FUNCTION F_Delete_ST_AnyType : HResult
VAR_INPUT
	name : STRING(80);
	varType : MPM_JsonParser.E_TypeClassEx;
END_VAR
VAR_IN_OUT
	stAnyType : MPM_JsonParser.ST_AnyType_User;
END_VAR
VAR
	pPointer_BYTE : POINTER TO BYTE;
	pPointer_BOOL : POINTER TO BOOL;
	pPointer_LREAL : POINTER TO LREAL;
	pPointer_DINT : POINTER TO DINT;
	pPointer_LINT : POINTER TO LINT;	
	pPointer_UDINT : POINTER TO UDINT;	
	pPointer_INT : POINTER TO INT;		
	pPointer_REAL : POINTER TO REAL;
	pPointer_WORD : POINTER TO WORD;		
END_VAR

stAnyType.name := name;
stAnyType.typeclass := varType;
IF stAnyType.pvalue > 0 THEN
	F_Delete_ST_AnyType := MPM_FBResult.E_Result.S_FAILED;
	RETURN;
END_IF
CASE varType OF
	MPM_JsonParser.E_TypeClassEx.TYPE_BOOL:
		pPointer_BYTE := stAnyType.pvalue;
		stAnyType.diSize := SIZEOF(BOOL);
		F_Delete_ST_AnyType := MPM_FBResult.E_Result.S_OK;
	MPM_JsonParser.E_TypeClassEx.TYPE_BYTE:
		stAnyType.pvalue := __NEW(BYTE);	
		stAnyType.diSize := SIZEOF(BYTE);	
		F_Delete_ST_AnyType := MPM_FBResult.E_Result.S_OK;
	MPM_JsonParser.E_TypeClassEx.TYPE_LREAL:
		stAnyType.pvalue := __NEW(LREAL);	
		stAnyType.diSize := SIZEOF(LREAL);	
		F_Delete_ST_AnyType := MPM_FBResult.E_Result.S_OK;		
	MPM_JsonParser.E_TypeClassEx.TYPE_DINT:
		stAnyType.pvalue := __NEW(DINT);	
		stAnyType.diSize := SIZEOF(DINT);	
		F_Delete_ST_AnyType := MPM_FBResult.E_Result.S_OK;
	MPM_JsonParser.E_TypeClassEx.TYPE_LINT:
		stAnyType.pvalue := __NEW(LINT);	
		stAnyType.diSize := SIZEOF(LINT);
		F_Delete_ST_AnyType := MPM_FBResult.E_Result.S_OK;	
	MPM_JsonParser.E_TypeClassEx.TYPE_UDINT:
		stAnyType.pvalue := __NEW(UDINT);	
		stAnyType.diSize := SIZEOF(UDINT);
		F_Delete_ST_AnyType := MPM_FBResult.E_Result.S_OK;	
	MPM_JsonParser.E_TypeClassEx.TYPE_INT:
		stAnyType.pvalue := __NEW(INT);	
		stAnyType.diSize := SIZEOF(INT);
		F_Delete_ST_AnyType := MPM_FBResult.E_Result.S_OK;		
	MPM_JsonParser.E_TypeClassEx.TYPE_REAL:
		stAnyType.pvalue := __NEW(REAL);	
		stAnyType.diSize := SIZEOF(REAL);	
		F_Delete_ST_AnyType := MPM_FBResult.E_Result.S_OK;		
	MPM_JsonParser.E_TypeClassEx.TYPE_WORD:
		stAnyType.pvalue := __NEW(WORD);	
		stAnyType.diSize := SIZEOF(WORD);	
		F_Delete_ST_AnyType := MPM_FBResult.E_Result.S_OK;		
	ELSE
		F_Delete_ST_AnyType := MPM_FBResult.E_Result.S_FAILED;				
END_CASE

END_FUNCTION

(* stored: Version 1.1.0.1, ProductVersion 3.1.4024.12
   POU F_Delete_ST_AnyType: Id {4d1f2cd0-f10f-4f75-b58a-0c6d643a48ea}, SpecialFunc None *)
